TYPE ST_PlanarObjectInfoEx EXTENDS Tc3_Mc3PlanarMotion.PlanarObjectInfo :
STRUCT
	ipObject : I_CH_Object;
END_STRUCT
END_TYPE

(* stored: Version 1.1.0.1, ProductVersion 3.1.4024.12
   DUT ST_PlanarObjectInfoEx: Id {e7c03c06-7a8e-4563-b3e3-964ea6e243a7} *)
